KUKA KRL program: art_placepoint.src, art_placepoint.dat

--- art_placepoint.src ---
&ACCESS RVO2
&REL 57
&PARAM EDITMASK = *
&PARAM TEMPLATE = C:\KRC\Roboter\Template\vorgabe
&PARAM DISKPATH = KRC:\R1\TP\ART
DEF art_placepoint ( )
END
;
; Work area init.
;
GLOBAL DEF ART_PP_Initialize()
   DECL INT line_num
   DECL INT place_point_num
   FOR line_num = 1 TO DEF_LINE_COUNT
      FOR place_point_num = 1 TO 1
         ART_place_point[line_num, place_point_num].state = #WA_IN
         ART_place_point[line_num, place_point_num].passed = FALSE
         ART_place_point[line_num, place_point_num].pallet_out = FALSE
         ART_place_point[line_num, place_point_num].buttonPressTime = 0
         ART_place_point[line_num, place_point_num].error_state = #NORMAL

         ;ART_work_areas[chain_num, place_point_num].scheme_number = 0
         ARTHMIClearMessage(ART_place_point[line_num, place_point_num].m_handle_not_ready)
         ARTHMIClearMessage(ART_place_point[line_num, place_point_num].m_h_service_mode)
         ARTHMIClearMessage(ART_place_point[line_num, place_point_num].m_h_barrier_pass)
         ARTHMIClearMessage(ART_place_point[line_num, place_point_num].m_handle_ready_conf)
         ARTHMIClearMessage(ART_place_point[line_num, place_point_num].m_pallet_out)
      ENDFOR
   ENDFOR

END
;
; Select ready work area.
;
GLOBAL DEF ART_PP_Select()
   DECL INT line_num
   DECL INT place_point_num
   FOR line_num = 1 TO DEF_LINE_COUNT
      ; Continue when work area selected
      IF (ART_line[line_num].useWorkArea <= 0) THEN
         ; Select ready work area
         FOR place_point_num = 1 TO DEF_WA_COUNT
            IF (ART_place_point[line_num, place_point_num].state == #WA_READY) THEN
               ART_line[line_num].useWorkArea = place_point_num
               ART_line_new_scheme(line_num)
            ENDIF
         ENDFOR
      ENDIF
      IF (ART_line[line_num].useWorkArea > 0) THEN
         ART_place_point[line_num, ART_line[line_num].useWorkArea].state = #WA_BUSY
      ENDIF
   ENDFOR
END
;
; Reset BUSY state, when scheme changed. After select ready work area.
;
GLOBAL DEF ART_PP_sheme_changed()
   DECL INT line_num
   DECL INT place_point_num
   FOR line_num = 1 TO DEF_LINE_COUNT
      IF ART_line[line_num].scheme_change THEN
         FOR place_point_num = 1 TO DEF_WA_COUNT
            IF (ART_place_point[line_num, place_point_num].state == #WA_BUSY) THEN
               ART_line[line_num].scheme_change = FALSE
               ART_PP_Full(line_num)
            ENDIF
         ENDFOR
      ENDIF
   ENDFOR

   ART_PP_Select()
END
;
; Set work area to full state.
;
GLOBAL DEF ART_PP_Full(line_num: IN)
   DECL INT line_num
   ART_place_point[line_num, ART_line[line_num].useWorkArea].state = #WA_OUT
   ART_line[line_num].isPalletDone = FALSE
   ART_line[line_num].is50PercentDone = FALSE
   ART_line[line_num].current_bag = 0
   ART_line[line_num].useWorkArea = 0
END
;
; Work area pallet out.
;
GLOBAL DEF ART_PP_pallet_out(line_num :IN, place_point_num :IN)
   DECL INT line_num
   DECL INT place_point_num

   ;IF (ART_work_areas[line_num, place_point_num].state == #WA_OUT) THEN
   ART_place_point[line_num, place_point_num].state = #WA_GIVE_WAIT
   ;ENDIF
END
;
; Work area pallet in.
;
GLOBAL DEF ART_PP_pallet_in(line_num :IN, place_point_num :IN)
   DECL INT line_num
   DECL INT place_point_num

   IF (ART_place_point[line_num, place_point_num].state == #WA_IN) THEN
      ART_place_point[line_num, place_point_num].state = #WA_READY
   ENDIF
END
;
; Work areas SPS.
;
GLOBAL DEF ART_PP_DoSPS()
   DECL INT line_num
   DECL INT place_point_num
   ;
   ; var binding
   ;

   ART_place_point[1,1].di_FramePalletIn = diConveyor8Out
   ART_place_point[2,1].di_FramePalletIn = diConveyor9Out

   FOR line_num = 1 TO DEF_LINE_COUNT
      FOR place_point_num = 1 TO DEF_WA_COUNT
         IF ARTHMIIsResetPushed() THEN
            ART_place_point[line_num, place_point_num].error_state = #NORMAL
         ENDIF
         ;
         ; Wait pallet giving state.
         ;
         IF (ART_place_point[line_num, place_point_num].state == #WA_GIVE_WAIT) THEN
             IF ARTDispencerGive() THEN
                ART_place_point[line_num, place_point_num].state = #WA_IN
             ENDIF
         ENDIF
         ;
         ; IN state.
         ;
         IF (ART_place_point[line_num, place_point_num].state == #WA_IN) THEN
            IF ART_place_point[line_num, place_point_num].di_FramePalletIn THEN
               ART_place_point[line_num, place_point_num].state = #WA_READY
            ENDIF
         ENDIF
         ;
         ; READY state.
         ;
         IF (ART_place_point[line_num, place_point_num].state == #WA_READY) THEN
             IF ARTDispencerGive() THEN
                ART_place_point[line_num, place_point_num].state = #WA_IN
             ENDIF
         ENDIF
         ;
         ; BUSY state.
         ;
         IF (ART_place_point[line_num, place_point_num].state == #WA_BUSY) THEN
            IF NOT ART_place_point[line_num, place_point_num].di_FramePalletIn THEN
               ARTHMISetMessage(ART_place_point[line_num, place_point_num].m_pallet_out, TRUE, "ARTWA", "WA_PALLET_OUT")
               ART_place_point[line_num, place_point_num].error_state = #ERROR
               ARTSystemSetState(#ARTSYS_STATE_ERROR)
            ENDIF
         ENDIF
         ;
         ; OUT state.
         ;
         IF (ART_place_point[line_num, place_point_num].state == #WA_OUT) THEN
         ENDIF

      ENDFOR
   ENDFOR
   ;
   ; Test
   ;
   IF doTest_WA1_Full THEN
      ART_PP_Full(1)
      doTest_WA1_Full = FALSE
   ENDIF
   IF doTest_WA2_Full THEN
      ART_PP_Full(2)
      doTest_WA2_Full = FALSE
   ENDIF
END

--- art_placepoint.dat ---
&ACCESS RVO2
&REL 57
&PARAM EDITMASK = *
&PARAM TEMPLATE = C:\KRC\Roboter\Template\vorgabe
&PARAM DISKPATH = KRC:\R1\TP\ART
DEFDAT  art_placepoint PUBLIC
GLOBAL ENUM ART_PP_STATES WA_BUSY,WA_FULL,WA_READY,WA_IN,WA_OUT,WA_SERVICE,WA_OPERATOR,WA_GIVE_WAIT
GLOBAL STRUC PLACE_POINT ART_PP_STATES state, ART_DEVICE_STATE error_state,BOOL isFramePalletEvro,BOOL do_safety_mute,BOOL do_blink,BOOL di_barrier_pass,BOOL di_ready_button,BOOL di_FramePalletIn,BOOL di_FrameHasBags,BOOL isServiceModeOff,INT buttonPressTime,BOOL ready_signal,BOOL ready_canceled,INT m_h_wrong_pallet,INT m_h_barrier_pass,INT m_handle_ready_conf,INT m_handle_not_ready,INT m_h_service_mode,BOOL do_ready_button_lamp,BOOL passed,BOOL pallet_out,INT m_pallet_out
DECL INT DEF_WA_COUNT=1
DECL GLOBAL PLACE_POINT ART_place_point[2,2]
;DECL GLOBAL INT ART_WA_useWorkArea[2]
;DECL GLOBAL INT ART_WA_new_scheme[2]
; Chain 1
ART_place_point[1,1]={state #WA_BUSY,error_state #NORMAL,isFramePalletEvro TRUE,do_safety_mute TRUE,do_blink FALSE,di_barrier_pass FALSE,di_ready_button FALSE,di_FramePalletIn TRUE,di_FrameHasBags FALSE,isServiceModeOff TRUE,buttonPressTime 0,ready_signal FALSE,ready_canceled FALSE,m_h_wrong_pallet 0,m_h_barrier_pass 0,m_handle_ready_conf 0,m_handle_not_ready 0,m_h_service_mode 0,do_ready_button_lamp FALSE,passed FALSE,pallet_out FALSE,m_pallet_out 0}
ART_place_point[1,2]={state #WA_BUSY,error_state #NORMAL,isFramePalletEvro FALSE,do_safety_mute FALSE,do_blink FALSE,di_barrier_pass FALSE,di_ready_button FALSE,di_FramePalletIn FALSE,di_FrameHasBags FALSE,isServiceModeOff TRUE,buttonPressTime 0,ready_signal FALSE,ready_canceled FALSE,m_h_wrong_pallet 0,m_h_barrier_pass 0,m_handle_ready_conf 0,m_handle_not_ready 0,m_h_service_mode 0,do_ready_button_lamp TRUE,passed FALSE,pallet_out FALSE,m_pallet_out 0}
;ART_WA_useWorkArea[1]=0
;ART_WA_new_scheme[1]=1
; Chain 2
;ART_work_areas[2,1]={state #WA_BUSY,isFramePalletEvro TRUE,do_safety_mute FALSE,do_blink FALSE,di_barrier_pass FALSE,di_ready_button FALSE,di_FramePalletIn TRUE,di_FrameHasBags TRUE,isServiceModeOff TRUE,buttonPressTime 0,ready_signal FALSE,ready_canceled FALSE,m_h_wrong_pallet 0,m_h_barrier_pass 0,m_handle_ready_conf 0,m_handle_not_ready 0,m_h_service_mode 0,do_ready_button_lamp TRUE,passed FALSE,pallet_out FALSE,m_pallet_out 0}
;ART_work_areas[2,2]={state #WA_OPERATOR,isFramePalletEvro FALSE,do_safety_mute TRUE,do_blink FALSE,di_barrier_pass FALSE,di_ready_button FALSE,di_FramePalletIn FALSE,di_FrameHasBags FALSE,isServiceModeOff TRUE,buttonPressTime 0,ready_signal FALSE,ready_canceled FALSE,m_h_wrong_pallet 0,m_h_barrier_pass 0,m_handle_ready_conf 0,m_handle_not_ready 0,m_h_service_mode 0,do_ready_button_lamp FALSE,passed FALSE,pallet_out FALSE,m_pallet_out 0}
;ART_WA_useWorkArea[2]=0
;ART_WA_new_scheme[2]=1

DECL CONST INT BUTTON_PRESS_TIME=1000
; Log
DECL INT ART_WA_OperWaitTimer=644977708
DECL GLOBAL INT ART_WA_OperWaitTime=200
DECL GLOBAL BOOL ART_WA_OperWaitTimeF=TRUE
DECL INT ART_WA_PalletChgTimer=0
DECL GLOBAL INT ART_WA_PalletChgTime=227
DECL GLOBAL BOOL ART_WA_PalletChgTimeF=TRUE

ENDDAT
